{attribute addProperty BoxType "EL6201-0000-0017"}
{attribute addProperty Id "Slave_21A_DI0BIT10.125161Slave_21A_DI1BIT10.125162Slave_21A_DI2BIT10.125163Slave_21A_DI3BIT10.125164Slave_21B_DI0BIT10.125165Slave_21B_DI1BIT10.125166Slave_21B_DI2BIT10.125167Slave_21B_DI3BIT10.125168"}
{attribute addProperty CRC "3386450094"}
{attribute addProperty SizeInBites "8"}
{attribute addProperty SizeInBytes "1"}
TYPE Slave_21_Inputs_C9D920AE :
STRUCT
	{attribute addProperty Name "Slave_21A_DI0"}
	Slave_21A_DI0 : BIT;
	{attribute addProperty Name "Slave_21A_DI1"}
	Slave_21A_DI1 : BIT;
	{attribute addProperty Name "Slave_21A_DI2"}
	Slave_21A_DI2 : BIT;
	{attribute addProperty Name "Slave_21A_DI3"}
	Slave_21A_DI3 : BIT;
	{attribute addProperty Name "Slave_21B_DI0"}
	Slave_21B_DI0 : BIT;
	{attribute addProperty Name "Slave_21B_DI1"}
	Slave_21B_DI1 : BIT;
	{attribute addProperty Name "Slave_21B_DI2"}
	Slave_21B_DI2 : BIT;
	{attribute addProperty Name "Slave_21B_DI3"}
	Slave_21B_DI3 : BIT;
END_STRUCT
END_TYPE

(* stored: Version 1.2.0.0, ProductVersion 3.1.4024.9
   DUT Slave_21_Inputs_C9D920AE: Id {6739268c-caa5-4557-aa62-cc9ff256953b} *)
